Staubli VAL3: onF3Event.pgx

program onF3Event()
  local string l_sMessage
  local bool l_bInside
begin
  // look if the bButton is enable
  if bButton[2]
    //
    // go to next POINT
    //
    if !cycleStatus:bCycle or !cycleStatus:bSimulation
      // check for the point proximity
      call isAtPoint(nPoint,l_bInside)
      if l_bInside
        call goTo(nPoint+1)
      else
        call goTo(nPoint)
      endIf
    endIf
  endIf
end
